Staubli VAL3: LOADJOB.pgx

public program loadJob(num handle_, string value_, bool& result_[])
begin
  // load job from flash and make it active
  nCommand[handle_]=coLF
  call sendCommand(handle_,"lf"+value_,result_)
end
